(* CoDeSys 2.3.9.28 project: Aula06_furadeiraAutomatica.pro *)
(* Libraries: Standard.lib 27.1.09 11:27:38, Util.lib 27.1.09 11:27:38, IecSfc.lib*24.11.08 08:07:15, SysLibTime.lib*27.1.09 11:27:38, SysTaskInfo.lib 24.11.08 08:07:15, SYSLIBCALLBACK.LIB 27.1.09 11:27:38 *)

(* PLC configuration (modules and I/O channels)
Hexswitch AT %IB0 [HexSwitch] rotary switch 0 = STOP, 1-15 = RUN
IOModules [CPX_MASTER] node 0, in %IB4 out %QB0
  8DI/8DO [CPX-8DI_8DO_Multi_I_O_module_1] node 0, in %IB4 out %QB0 {StringParam = 4,8,1,8,1; ByteParam = 7; ByteParam = 81; ByteParam = 0; ByteParam = 0; ByteParam = 0; ByteParam = 0; ByteParam = 0; IdleStateParam = 0; IdleModeParam = 255; IdleStateParam = 0; IdleModeParam = 255; IdleStateParam = 0; IdleModeParam = 255; IdleStateParam = 0; IdleModeParam = 255}
    AT %IB4 [ByteInput] -
    AT %QB0 [ByteOutput] -
  8DI/8DO [CPX-8DI_8DO_Multi_I_O_module_1] node 1, in %IB8 out %QB4 {StringParam = 4,8,1,8,1; ByteParam = 7; ByteParam = 81; ByteParam = 0; ByteParam = 0; ByteParam = 0; ByteParam = 0; ByteParam = 0; IdleStateParam = 0; IdleModeParam = 255; IdleStateParam = 0; IdleModeParam = 255; IdleStateParam = 0; IdleModeParam = 255; IdleStateParam = 0; IdleModeParam = 255}
    AT %IB8 [ByteInput] -
    AT %QB4 [ByteOutput] -
*)

(* Global variable list: Global_Variables *)
VAR_GLOBAL

	START AT %IX2.0 : BOOL;
	S1 AT %IX2.1 : BOOL;
	S2 AT %IX2.2 : BOOL;
	S3 AT %IX2.3 : BOOL;
	STOP AT %IX2.4 : BOOL;

	C1 AT %QX0.0 : BOOL;
	C2 AT %QX0.1 : BOOL;
	M1 AT %QX0.2 : BOOL;
	LAMP AT %QX0.3 : BOOL;

	MEM1 : BOOL;

END_VAR

(* POU PLC_PRG, LD *)
PROGRAM PLC_PRG
VAR
END_VAR
VAR (* helpers for the ST form of the networks *)
	_p1 : BOOL;
END_VAR
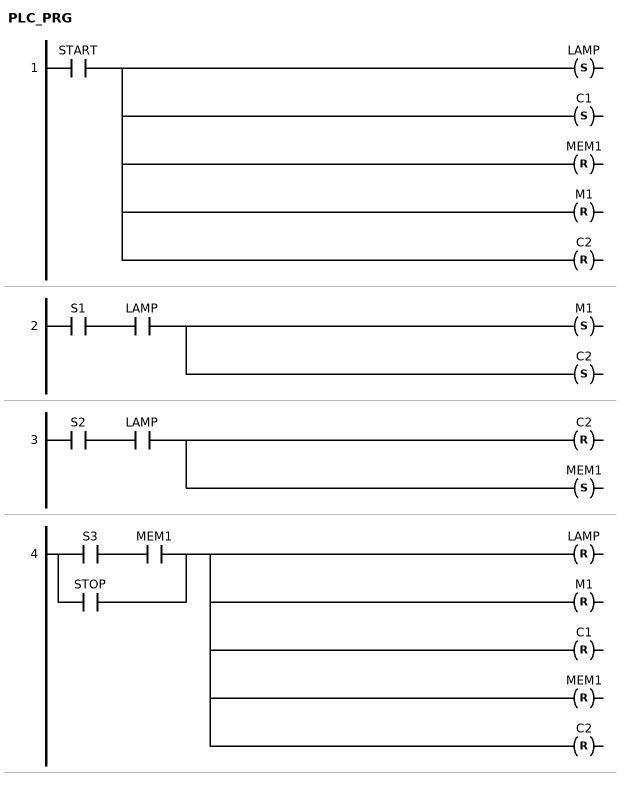
_LD_ (* Ladder Diagram *)
NETWORK 1
	[START] --- (S LAMP) (S C1) (R MEM1) (R M1) (R C2)
NETWORK 2
	[S1] - [LAMP] --- (S M1) (S C2)
NETWORK 3
	[S2] - [LAMP] --- (R C2) (S MEM1)
NETWORK 4
	{ [S3] - [MEM1] | [STOP] } --- (R LAMP) (R M1) (R C1) (R MEM1) (R C2)
_END_LD_
(* the same logic as Structured Text *)
(* Network 1 *)
IF START THEN LAMP := TRUE; C1 := TRUE; MEM1 := FALSE; M1 := FALSE; C2 := FALSE; END_IF;
(* Network 2 *)
IF S1 AND LAMP THEN M1 := TRUE; C2 := TRUE; END_IF;
(* Network 3 *)
IF S2 AND LAMP THEN C2 := FALSE; MEM1 := TRUE; END_IF;
(* Network 4 *)
_p1 := S3 AND MEM1 OR STOP;
IF _p1 THEN LAMP := FALSE; M1 := FALSE; C1 := FALSE; MEM1 := FALSE; C2 := FALSE; END_IF;
END_PROGRAM
